FUNCTION_BLOCK Example1WrappedComponent EXTENDS TcoCore.TcoComponent
VAR_INPUT
	inSignal: BOOL;
END_VAR
VAR_OUTPUT
END_VAR
VAR
		
      	piston : fbPiston(THIS^);
     	digitalInput : TcoDi(THIS^); 
     	digitaOutput : TcoDo(THIS^);
	
		dummy1Task : TcoCore.TcoTask(THIS^);
		dummy2Task : TcoCore.TcoTask(THIS^);
		Setpoint:INT;
END_VAR

piston();
digitalInput(inoSignal:=inSignal);

dummy1Task.Enabled:=TRUE;
IF dummy1Task.Execute() THEN
	;
END_IF

(*~
	<docu>
		<summary>
			Restores this instance to the Ready state. Can be called explicitly or from within one of the restore mechanisms.	
		</summary>			
	</docu>	
~*)
METHOD  Restore : ITcoRestorable
END_METHOD

(*~
	<docu>
		<summary>
		    Custom service (manual, maintenance) logic.
			This method must be implemented in derived class.
		</summary>			
	</docu>	
~*)
METHOD PROTECTED  ServiceMode
piston.Service();
digitalInput.Service();
digitaOutput.Service();
END_METHOD

END_FUNCTION_BLOCK

(* stored: Version 1.1.0.1
   POU Example1WrappedComponent: Id {d4287f36-2935-0b39-217a-2a1b69b3c8a2}, SpecialFunc None
   Method Restore: Id {38596799-d63f-0b45-099b-198ffa020014}
   Method ServiceMode: Id {7a71b670-599d-0eef-2aa3-3fa94a6f3779} *)
